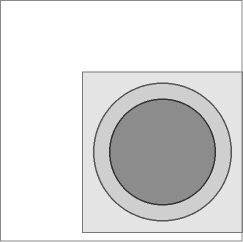
VISUALIZATION Visualization  // 243x242
    PushSwitch (82,62 161x180), variable: P_SerialCom.bStart, behaviour: TAP, style: Switch-PushSwitch-Gray
END_VISUALIZATION

(* stored: Version 1.1.0.1
   Visu Visualization: Id {5bd15c4b-ccf7-4061-954a-0818e71737bb} *)
